// Output from UI controller
// Input to master arm control task and cart control task  
TYPE ST_UIData :
STRUCT
	m_motionScale:LREAL := 1.0;
	m_faultClearFlag:BOOL := FALSE;
END_STRUCT
END_TYPE

(* stored: Version 1.1.0.1, ProductVersion 3.1.4024.12
   DUT ST_UIData: Id {80b16640-247c-4dd4-96a5-e4b5ddf546bb} *)
